ABB RAPID module: Module1.mod

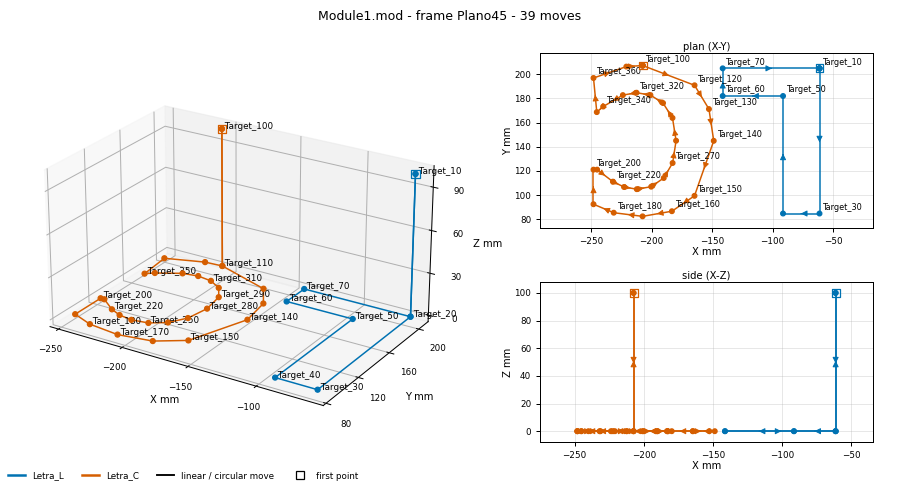
[picture p0: tool path of Module1.mod in frame Plano45, 39 of 41 moves have a stored position in this frame; points joined in program order, loops and branches not executed]
MODULE Module1
        CONST robtarget Target_10:=[[-61.252986291,204.835773881,99.999999785],[0,0.999944963,-0.010491487,0],[0,1,-2,0],[9E+09,9E+09,9E+09,9E+09,9E+09,9E+09]];
    CONST robtarget Target_20:=[[-61.252986291,204.835773777,-0.000000215],[0,0.999944963,-0.010491487,0],[0,2,-2,0],[9E+09,9E+09,9E+09,9E+09,9E+09,9E+09]];
    CONST robtarget Target_30:=[[-61.252986291,84.835773776,-0.000000089],[0,0.999944963,-0.010491487,0],[0,2,-2,0],[9E+09,9E+09,9E+09,9E+09,9E+09,9E+09]];
    CONST robtarget Target_40:=[[-91.39885339,84.835773776,-0.000000089],[0,0.999944963,-0.010491487,0],[0,2,-2,0],[9E+09,9E+09,9E+09,9E+09,9E+09,9E+09]];
    CONST robtarget Target_50:=[[-91.39885339,181.98326162,-0.000000191],[0,0.999944963,-0.010491487,0],[0,2,-2,0],[9E+09,9E+09,9E+09,9E+09,9E+09,9E+09]];
    CONST robtarget Target_60:=[[-141.285401202,181.98326162,-0.000000191],[0,0.999944963,-0.010491487,0],[0,1,-2,0],[9E+09,9E+09,9E+09,9E+09,9E+09,9E+09]];
    CONST robtarget Target_70:=[[-141.285401202,204.835773777,-0.000000215],[0,0.999944963,-0.010491487,0],[0,1,-2,0],[9E+09,9E+09,9E+09,9E+09,9E+09,9E+09]];
    CONST robtarget Target_80:=[[-61.252986291,204.835773777,-0.000000215],[0,0.999944963,-0.010491487,0],[0,2,-2,0],[9E+09,9E+09,9E+09,9E+09,9E+09,9E+09]];
    CONST robtarget Target_90:=[[-61.252986291,204.835773881,99.999999785],[0,0.999944963,-0.010491487,0],[0,1,-2,0],[9E+09,9E+09,9E+09,9E+09,9E+09,9E+09]];
    CONST robtarget Target_100:=[[-207.411819355,207.169647462,99.999999783],[0,0.999944963,-0.010491487,0],[0,1,-2,0],[9E+09,9E+09,9E+09,9E+09,9E+09,9E+09]];
    CONST robtarget Target_110:=[[-207.411819355,207.169647358,-0.000000217],[0,0.999944963,-0.010491487,0],[0,1,-2,0],[9E+09,9E+09,9E+09,9E+09,9E+09,9E+09]];
    CONST robtarget Target_120:=[[-164.526892288,190.832532285,-0.0000002],[0,0.999944963,-0.010491487,0],[0,1,-2,0],[9E+09,9E+09,9E+09,9E+09,9E+09,9E+09]];
    CONST robtarget Target_130:=[[-152.638723731,171.189096304,-0.00000018],[0.000000001,0.999944963,-0.010491487,0.000000001],[0,1,-2,0],[9E+09,9E+09,9E+09,9E+09,9E+09,9E+09]];
    CONST robtarget Target_140:=[[-148.676000878,144.933018508,-0.000000152],[0,0.999944963,-0.010491487,0],[0,2,-2,0],[9E+09,9E+09,9E+09,9E+09,9E+09,9E+09]];
    CONST robtarget Target_150:=[[-164.575514654,99.471106029,-0.000000104],[-0.000000001,0.999944963,-0.010491487,0],[0,2,-2,0],[9E+09,9E+09,9E+09,9E+09,9E+09,9E+09]];
    CONST robtarget Target_160:=[[-183.258658901,86.744201652,-0.000000091],[-0.000000001,0.999944963,-0.010491487,0],[0,2,-2,0],[9E+09,9E+09,9E+09,9E+09,9E+09,9E+09]];
    CONST robtarget Target_170:=[[-207.509064087,82.501900194,-0.000000087],[0,0.999944963,-0.010491487,0],[0,2,-2,0],[9E+09,9E+09,9E+09,9E+09,9E+09,9E+09]];
    CONST robtarget Target_180:=[[-231.334023568,85.516486904,-0.00000009],[-0.000000001,0.999944963,-0.010491487,0],[0,2,-2,0],[9E+09,9E+09,9E+09,9E+09,9E+09,9E+09]];
    CONST robtarget Target_190:=[[-248.060117572,92.51810765,-0.000000097],[-0.000000001,0.999944963,-0.010491487,0],[0,2,-2,0],[9E+09,9E+09,9E+09,9E+09,9E+09,9E+09]];
    CONST robtarget Target_200:=[[-248.060117572,121.108059027,-0.000000127],[0,0.999944963,-0.010491487,0],[0,1,-2,0],[9E+09,9E+09,9E+09,9E+09,9E+09,9E+09]];
    CONST robtarget Target_210:=[[-245.045530862,121.108059027,-0.000000127],[0,0.999944963,-0.010491487,0],[0,1,-2,0],[9E+09,9E+09,9E+09,9E+09,9E+09,9E+09]];
    CONST robtarget Target_220:=[[-232.014736696,111.189096305,-0.000000117],[0,0.999944963,-0.010491487,0.000000001],[0,2,-2,0],[9E+09,9E+09,9E+09,9E+09,9E+09,9E+09]];
    CONST robtarget Target_230:=[[-222.825109468,106.764460972,-0.000000112],[0,0.999944963,-0.010491487,0],[0,2,-2,0],[9E+09,9E+09,9E+09,9E+09,9E+09,9E+09]];
    CONST robtarget Target_240:=[[-212.274055983,104.965433419,-0.00000011],[0,0.999944963,-0.010491487,0],[0,2,-2,0],[9E+09,9E+09,9E+09,9E+09,9E+09,9E+09]];
    CONST robtarget Target_250:=[[-200.361576243,107.007572804,-0.000000112],[0.000000001,0.999944963,-0.010491487,0],[0,2,-2,0],[9E+09,9E+09,9E+09,9E+09,9E+09,9E+09]];
    CONST robtarget Target_260:=[[-190.005012223,114.203683014,-0.00000012],[0.000000001,0.999944963,-0.010491487,0],[0,2,-2,0],[9E+09,9E+09,9E+09,9E+09,9E+09,9E+09]];
    CONST robtarget Target_270:=[[-182.663034914,126.602386417,-0.000000133],[0.000000001,0.999944963,-0.010491487,-0.000000001],[0,2,-2,0],[9E+09,9E+09,9E+09,9E+09,9E+09,9E+09]];
    CONST robtarget Target_280:=[[-179.794315303,145.030263241,-0.000000152],[0,0.999944963,-0.010491487,0],[0,1,-2,0],[9E+09,9E+09,9E+09,9E+09,9E+09,9E+09]];
    CONST robtarget Target_290:=[[-182.760279646,163.847118995,-0.000000172],[-0.000000001,0.999944963,-0.010491487,-0.000000001],[0,1,-2,0],[9E+09,9E+09,9E+09,9E+09,9E+09,9E+09]];
    CONST robtarget Target_300:=[[-190.588480619,176.148577666,-0.000000185],[0,0.999944963,-0.010491487,0],[0,1,-2,0],[9E+09,9E+09,9E+09,9E+09,9E+09,9E+09]];
    CONST robtarget Target_310:=[[-200.993667004,182.712597115,-0.000000192],[-0.000000001,0.999944963,-0.010491487,0.000000001],[0,1,-2,0],[9E+09,9E+09,9E+09,9E+09,9E+09,9E+09]];
    CONST robtarget Target_320:=[[-212.468545449,184.706114133,-0.000000194],[0,0.999944963,-0.010491487,0],[0,1,-2,0],[9E+09,9E+09,9E+09,9E+09,9E+09,9E+09]];
    CONST robtarget Target_330:=[[-223.797556794,182.712597115,-0.000000192],[0,0.999944963,-0.010491487,0],[0,1,-2,0],[9E+09,9E+09,9E+09,9E+09,9E+09,9E+09]];
    CONST robtarget Target_340:=[[-240.037427134,173.279858055,-0.000000182],[0,0.999944963,-0.010491487,0],[0,1,-2,0],[9E+09,9E+09,9E+09,9E+09,9E+09,9E+09]];
    CONST robtarget Target_350:=[[-245.33726506,168.660733257,-0.000000177],[-0.000000001,0.999944963,-0.010491487,0],[0,1,-2,0],[9E+09,9E+09,9E+09,9E+09,9E+09,9E+09]];
    CONST robtarget Target_360:=[[-248.060117572,196.861705705,-0.000000206],[0,0.999944963,-0.010491487,0],[0,1,-2,0],[9E+09,9E+09,9E+09,9E+09,9E+09,9E+09]];
    CONST robtarget Target_370:=[[-220.880214816,206.294444764,-0.000000216],[0,0.999944963,-0.010491487,0],[0,1,-2,0],[9E+09,9E+09,9E+09,9E+09,9E+09,9E+09]];
    CONST robtarget Target_380:=[[-207.411819355,207.169647358,-0.000000217],[0,0.999944963,-0.010491487,0],[0,1,-2,0],[9E+09,9E+09,9E+09,9E+09,9E+09,9E+09]];
    CONST robtarget Target_390:=[[-207.411819355,207.169647462,99.999999783],[0,0.999944963,-0.010491487,0],[0,1,-2,0],[9E+09,9E+09,9E+09,9E+09,9E+09,9E+09]];
    CONST jointtarget MyHome_LC:=[[0,0,0,0,30,0],[9E+09,9E+09,9E+09,9E+09,9E+09,9E+09]];
    CONST jointtarget MyClose_LC:=[[0,25,20,170,15,-125],[9E+09,9E+09,9E+09,9E+09,9E+09,9E+09]];
!***********************************************************
    !
    ! Module:  Module1
    !
    ! Description:
    !   <Insert description here>
    !
    ! Author: user
    !
    ! Version: 1.0
    !
    !***********************************************************


    !***********************************************************
    !
    ! Procedure main
    !
    !   This is the entry point of your program
    !
    !***********************************************************
    PROC main()
        !Add your code here
        MyHomePath;
        MyClosePath;
        Letra_L;
        Letra_C;
        MyClosePath;
        MyHomePath;
    ENDPROC
    PROC Letra_L()
        MoveL Target_10,v200,z5,Marcador_LC\WObj:=Plano45;
        MoveL Target_20,v200,z5,Marcador_LC\WObj:=Plano45;
        MoveL Target_30,v200,z5,Marcador_LC\WObj:=Plano45;
        MoveL Target_40,v200,z5,Marcador_LC\WObj:=Plano45;
        MoveL Target_50,v200,z5,Marcador_LC\WObj:=Plano45;
        MoveL Target_60,v200,z5,Marcador_LC\WObj:=Plano45;
        MoveL Target_70,v200,z5,Marcador_LC\WObj:=Plano45;
        MoveL Target_80,v200,z5,Marcador_LC\WObj:=Plano45;
        MoveL Target_90,v200,z5,Marcador_LC\WObj:=Plano45;
    ENDPROC
    PROC Letra_C()
        MoveL Target_100,v200,z5,Marcador_LC\WObj:=Plano45;
        MoveL Target_110,v200,z5,Marcador_LC\WObj:=Plano45;
        MoveL Target_120,v200,z5,Marcador_LC\WObj:=Plano45;
        MoveL Target_130,v200,z5,Marcador_LC\WObj:=Plano45;
        MoveL Target_140,v200,z5,Marcador_LC\WObj:=Plano45;
        MoveL Target_150,v200,z5,Marcador_LC\WObj:=Plano45;
        MoveL Target_160,v200,z5,Marcador_LC\WObj:=Plano45;
        MoveL Target_170,v200,z5,Marcador_LC\WObj:=Plano45;
        MoveL Target_180,v200,z5,Marcador_LC\WObj:=Plano45;
        MoveL Target_190,v200,z5,Marcador_LC\WObj:=Plano45;
        MoveL Target_200,v200,z5,Marcador_LC\WObj:=Plano45;
        MoveL Target_210,v200,z5,Marcador_LC\WObj:=Plano45;
        MoveL Target_220,v200,z5,Marcador_LC\WObj:=Plano45;
        MoveL Target_230,v200,z5,Marcador_LC\WObj:=Plano45;
        MoveL Target_240,v200,z5,Marcador_LC\WObj:=Plano45;
        MoveL Target_250,v200,z5,Marcador_LC\WObj:=Plano45;
        MoveL Target_260,v200,z5,Marcador_LC\WObj:=Plano45;
        MoveL Target_270,v200,z5,Marcador_LC\WObj:=Plano45;
        MoveL Target_280,v200,z5,Marcador_LC\WObj:=Plano45;
        MoveL Target_290,v200,z5,Marcador_LC\WObj:=Plano45;
        MoveL Target_300,v200,z5,Marcador_LC\WObj:=Plano45;
        MoveL Target_310,v200,z5,Marcador_LC\WObj:=Plano45;
        MoveL Target_320,v200,z5,Marcador_LC\WObj:=Plano45;
        MoveL Target_330,v200,z5,Marcador_LC\WObj:=Plano45;
        MoveL Target_340,v200,z5,Marcador_LC\WObj:=Plano45;
        MoveL Target_350,v200,z5,Marcador_LC\WObj:=Plano45;
        MoveL Target_360,v200,z5,Marcador_LC\WObj:=Plano45;
        MoveL Target_370,v200,z5,Marcador_LC\WObj:=Plano45;
        MoveL Target_380,v200,z5,Marcador_LC\WObj:=Plano45;
        MoveL Target_390,v200,z5,Marcador_LC\WObj:=Plano45;
    ENDPROC
    PROC MyHomePath()
        MoveAbsJ MyHome_LC,v200,z5,Marcador_LC\WObj:=Plano45;
    ENDPROC
    PROC MyClosePath()
        MoveAbsJ MyClose_LC,v200,z5,Marcador_LC\WObj:=Plano45;
    ENDPROC
ENDMODULE
